(* IEC 61131-3 sources: ax-factoryio-assembler/src/ControlModules, 6 files *)

(* ---- ModeSwitch.st ---- *)
TYPE
    OperationMode : (Manual, Auto);
END_TYPE

NAMESPACE Demo.ControlModule
CLASS ModeSwitch IMPLEMENTS ICyclic
    VAR PUBLIC
        ModeSignal: REF_TO BOOL;
    END_VAR

    VAR PROTECTED
        _mode: OperationMode;
    END_VAR

    METHOD PUBLIC GetOperationMode: OperationMode
        GetOperationMode := _mode;
    END_METHOD

    METHOD PUBLIC Cycle
        IF ModeSignal^ THEN
            _mode := OperationMode#Auto;
        ELSE
            _mode := OperationMode#Manual;
        END_IF;
    END_METHOD
END_CLASS
END_NAMESPACE

(* ---- Clamp.st ---- *)
NAMESPACE Demo.ControlModule

INTERFACE IClamp EXTENDS ICyclic
    METHOD DoClamp
    END_METHOD

    METHOD Release
    END_METHOD

    METHOD Raise
    END_METHOD

    METHOD Down
    END_METHOD

    METHOD Reset
    END_METHOD
END_INTERFACE

CLASS Clamp IMPLEMENTS IClamp
    VAR PROTECTED
        _clampCmd: BOOL;
        _raiseCmd: BOOL;
    END_VAR

    VAR PUBLIC
        ClampedSignal: REF_TO BOOL;
        ClampSignal: REF_TO BOOL;
        RaiseSignal: REF_TO BOOL;
    END_VAR

    METHOD PUBLIC DoClamp
        _clampCmd := TRUE;
    END_METHOD

    METHOD PUBLIC Release
        _clampCmd := FALSE;
    END_METHOD

    METHOD PUBLIC Raise
        _raiseCmd := TRUE;
    END_METHOD

    METHOD PUBLIC Down
        _raiseCmd := FALSE;
    END_METHOD

    METHOD PUBLIC Reset
        _raiseCmd := FALSE;
        _clampCmd := FALSE;
    END_METHOD

    METHOD PUBLIC Cycle
        ClampSignal^ := _clampCmd;
        RaiseSignal^ := _raiseCmd;
    END_METHOD
END_CLASS
END_NAMESPACE

(* ---- Conveyor.st ---- *)
USING System.Timer;
NAMESPACE Demo.ControlModule

INTERFACE IConveyor EXTENDS ICyclic
    METHOD Start
    END_METHOD

    METHOD Stop
    END_METHOD
END_INTERFACE

CLASS Conveyor IMPLEMENTS IConveyor
    VAR PROTECTED
        _isOn : BOOL;
    END_VAR

    VAR PUBLIC
        ControlSignal: REF_TO BOOL;
    END_VAR

    METHOD PUBLIC Start
        _isOn := TRUE;
    END_METHOD

    METHOD PUBLIC Stop
        _isOn := FALSE;
    END_METHOD

    METHOD PUBLIC Cycle
        ControlSignal^ := _isOn;
    END_METHOD
END_CLASS
END_NAMESPACE

(* ---- Sensor.st ---- *)
NAMESPACE Demo.ControlModule

INTERFACE IObjectSensor EXTENDS ICyclic
    METHOD HasObjectPassed : BOOL
    END_METHOD

    METHOD Reset
    END_METHOD
END_INTERFACE

CLASS ObjectSensor IMPLEMENTS IObjectSensor
    VAR PROTECTED
        _hasObjectPassed: BOOL;
    END_VAR

    VAR PUBLIC
        ObjectDetectedInput: REF_TO BOOL;
    END_VAR

    METHOD PUBLIC HasObjectPassed : BOOL
        HasObjectPassed := _hasObjectPassed;
    END_METHOD

    METHOD PUBLIC Reset
        _hasObjectPassed :=FALSE;
    END_METHOD

    METHOD PUBLIC Cycle
        _hasObjectPassed :=  _hasObjectPassed | objectDetectedInput^;
    END_METHOD
END_CLASS
END_NAMESPACE

(* ---- Button.st ---- *)
NAMESPACE Demo.ControlModule
CLASS PUBLIC Button IMPLEMENTS ICyclic
    VAR PUBLIC
        Signal: REF_TO BOOL;
        HMI: REF_TO BOOL;
    END_VAR

    METHOD PUBLIC IsPressed : BOOL
        IF HMI <> NULL THEN
            IsPressed := Signal^ OR HMI^;
        ELSE
            IsPressed := Signal^;
        END_IF;
    END_METHOD

    METHOD PUBLIC Cycle
        ;
    END_METHOD
END_CLASS
END_NAMESPACE

(* ---- ButtotWithLight.st ---- *)
NAMESPACE Demo.ControlModule
CLASS ButtonWithLight EXTENDS Button IMPLEMENTS ICyclic
    VAR PUBLIC
        LightSignal: REF_TO BOOL;
    END_VAR

    METHOD PUBLIC OVERRIDE Cycle
        LightSignal^ := Signal^;
    END_METHOD
END_CLASS
END_NAMESPACE
